{attribute addProperty BoxType "EL3783-0000-0018"}
{attribute addProperty Id "L1_Voltage_StatusAT %I*L1_Voltage_Status_C389D43D1620L1_Voltage_SamplesAT %I*L1_Voltage_Samples_659DFAC6320400L1_Current_StatusAT %I*L1_Current_Status_507DE7B31620L1_Current_SamplesAT %I*L1_Current_Samples_41B62C85320400L2_Voltage_StatusAT %I*L2_Voltage_Status_F072DF281620L2_Voltage_SamplesAT %I*L2_Voltage_Samples_143DBB33320400L2_Current_StatusAT %I*L2_Current_Status_6386ECA61620L2_Current_SamplesAT %I*L2_Current_Samples_30166D70320400L3_Voltage_StatusAT %I*L3_Voltage_Status_1D64D2B61620L3_Voltage_SamplesAT %I*L3_Voltage_Samples_3B5D8460320400L3_Current_StatusAT %I*L3_Current_Status_8E90E1381620L3_Current_SamplesAT %I*L3_Current_Samples_1F765223320400AI_NextSync1TimeAT %I*AI_NextSync1Time_54B31DA16480AI_Sample_CountAT %I*AI_Sample_Count_46F3E31D1620AI_Current_RangeAT %I*AI_Current_Range_716B32064050WcStateAT %I*WcState_98A4DF7520.250InfoDataAT %I*InfoData_0BDED7BF144180"}
{attribute addProperty CRC "2863768150"}
{attribute addProperty SizeInBites "2282"}
{attribute addProperty SizeInBytes "285.25"}
TYPE EL3783_81B4F671 :
STRUCT
	{attribute addProperty Name "L1_Voltage_Status"}
	L1_Voltage_Status : L1_Voltage_Status_C389D43D;
	{attribute addProperty Name "L1_Voltage_Samples"}
	L1_Voltage_Samples : L1_Voltage_Samples_659DFAC6;
	{attribute addProperty Name "L1_Current_Status"}
	L1_Current_Status : L1_Current_Status_507DE7B3;
	{attribute addProperty Name "L1_Current_Samples"}
	L1_Current_Samples : L1_Current_Samples_41B62C85;
	{attribute addProperty Name "L2_Voltage_Status"}
	L2_Voltage_Status : L2_Voltage_Status_F072DF28;
	{attribute addProperty Name "L2_Voltage_Samples"}
	L2_Voltage_Samples : L2_Voltage_Samples_143DBB33;
	{attribute addProperty Name "L2_Current_Status"}
	L2_Current_Status : L2_Current_Status_6386ECA6;
	{attribute addProperty Name "L2_Current_Samples"}
	L2_Current_Samples : L2_Current_Samples_30166D70;
	{attribute addProperty Name "L3_Voltage_Status"}
	L3_Voltage_Status : L3_Voltage_Status_1D64D2B6;
	{attribute addProperty Name "L3_Voltage_Samples"}
	L3_Voltage_Samples : L3_Voltage_Samples_3B5D8460;
	{attribute addProperty Name "L3_Current_Status"}
	L3_Current_Status : L3_Current_Status_8E90E138;
	{attribute addProperty Name "L3_Current_Samples"}
	L3_Current_Samples : L3_Current_Samples_1F765223;
	{attribute addProperty Name "AI_NextSync1Time"}
	AI_NextSync1Time : AI_NextSync1Time_54B31DA1;
	{attribute addProperty Name "AI_Sample_Count"}
	AI_Sample_Count : AI_Sample_Count_46F3E31D;
	{attribute addProperty Name "AI_Current_Range"}
	AI_Current_Range : AI_Current_Range_716B3206;
	{attribute addProperty Name "WcState"}
	WcState : WcState_98A4DF75;
	{attribute addProperty Name "InfoData"}
	InfoData : InfoData_0BDED7BF;
END_STRUCT
END_TYPE

(* stored: Version 1.2.0.0, ProductVersion 3.1.4024.9
   DUT EL3783_81B4F671: Id {868883aa-c5bc-4ce0-877c-af308603ee0f} *)
